// TwinCAT 3 PLC project rixs_optics
// ProgramVersion: 3.1.4022.7
// libraries:
//   lcls2-cc-lib, * (SLAC)
//   PMPS, * (SLAC - LCLS)
//   Tc2_MC2, * (Beckhoff Automation GmbH)
//   Tc2_SerialCom, * (Beckhoff Automation GmbH)
//   Tc2_Standard, * (Beckhoff Automation GmbH)
//   Tc2_System, * (Beckhoff Automation GmbH)
//   Tc2_TcpIp, * (Beckhoff Automation GmbH)
//   Tc2_Utilities, * (Beckhoff Automation GmbH)
//   Tc3_Module, * (Beckhoff Automation GmbH)
//   LCLS General,newest,SLAC
//   lcls-twincat-motion,newest,SLAC
//   lcls-twincat-optics,newest,SLAC
// project tree:
//   DUTs/ ENUM_XS_YAG_States.TcDUT (not stored)
//   Function Blocks/ FB_XS_YAG_States.TcPOU (not stored)
//   GVLs/ GVL_COM_Buffers.TcGVL (not stored), GVL_M1K1.TcGVL (not stored), GVL_M1K1_BENDER_Constants.TcGVL (not stored), GVL_M1K1_BENDER_RTD.TcGVL (not stored), GVL_M1K1_Constants.TcGVL (not stored), GVL_M1K2.TcGVL (not stored), GVL_M1K2_Constants.TcGVL (not stored), GVL_PMPS.TcGVL (not stored), GVL_SerialIO.TcGVL (not stored), Main.TcGVL (not stored)
//   / PiezoDriver.TcTTO (not stored), PlcTask.TcTTO (not stored), SerialIO.TcTTO (not stored)
//   POUs/DAQ Comm/ DUT_01_Channel_NW.TcDUT (not stored), DUT_Channel_NW.TcDUT (not stored), DUT_Header_NW.TcDUT (not stored), FB_AssembleChannel.TcPOU (not stored), FB_AssembleHeader.TcPOU (not stored), FB_UDPSocketHandler.TcPOU (not stored), F_AddChannelToHeader.TcPOU (not stored)
//   POUs/ PRG_1_PlcTask.TcPOU (not stored), PRG_2_PMPS_POST.TcPOU (not stored), PRG_DAQ_ENCODER.TcPOU (not stored), PRG_MR1K1_BEND.TcPOU (not stored), PRG_MR1K1_BEND_BENDER.TcPOU (not stored), PRG_MR1K2_SWITCH.TcPOU (not stored), PRG_SL1K2_EXIT.TcPOU (not stored), PRG_SP1K1_MONO.TcPOU (not stored), PRG_SPO_PMPS.TcPOU (not stored), PRG_ST1K1_ZOS.TcPOU (not stored), PRG_ZeroOrder_PMPS.TcPOU
//   POUs/Serial Comm/ PiezoSerial.TcPOU (not stored), P_Serial_Com.TcPOU (not stored)
//   Zero Order Functions/ Zbm3.TcPOU, hbm3.TcPOU, Theta_m3.TcPOU

// ---- POUs/PRG_ZeroOrder_PMPS.TcPOU
PROGRAM PRG_ZeroOrder_PMPS
VAR
END_VAR

END_PROGRAM

// ---- Zero Order Functions/Zbm3.TcPOU
FUNCTION Zbm3 : REAL
VAR_INPUT
END_VAR
VAR
END_VAR

END_FUNCTION

// ---- Zero Order Functions/hbm3.TcPOU
FUNCTION hbm3 : REAL
VAR_INPUT
	Zbm: REAL;
END_VAR
VAR
	Pm3 : REAL;
	Hm3 : REAL;
END_VAR
VAR CONSTANT
	Zpiv : REAL:= 739.622 ; //m
	Hpiv : REAL:= 1.621305;//1.620305 + 0.001 // m 0.001 is correction from nominal
END_VAR


//Pm3 = mono grating pitch - 63300 urad
Pm3 := Main.M7.fPosition - 63300;

//hm3 = Hpiv + 0.006 m
Hm3 :=  Hpiv + 0.006;


hbm3 := TAN(Pm3) * Zbm + Hm3 - TAN(Pm3)*Zpiv;

END_FUNCTION

// ---- Zero Order Functions/Theta_m3.TcPOU
FUNCTION Theta_m3 : REAL
VAR_INPUT
END_VAR
VAR
	Pm3 : REAL;
	Pm2: REAL;
	Pm1: REAL;
	Theta0 : REAL:=0;
END_VAR



//Pm3 = mono grating pitch - 63300 urad
Pm3 := Main.M7.fPosition - 63300;

//Pm2 = mono mirror pitch - 90700 urad
Pm2 := Main.M6.fPosition - 90700;

//Pm1 = 18310 - 281 + mr1k1 bend pitch 
Pm1 := 18310 - 281 + Main.M16.fPosition;

Theta_m3 := 2 *Pm3 - 2 * Pm2 + 2* Pm1 - Theta0;

END_FUNCTION
